PROGRAM RTClock
VAR
	fbGetLocalTime  	: NT_GetTime;
	bBusy				: BOOL;
	bError          	: BOOL :=FALSE;
	nErrID          	: UDINT;
	presetTime      	: TIMESTRUCT;
	syncTimer       	: TON;
	syncTrigger     	: F_TRIG;
	bSynchronize		: BOOL;
	fbRTC_EX2       	: RTC_EX2;
	nMicroseconds   	: DWORD;
	sNetId 				:STRING := '172.16.5.8.1.1';
	LokalClock: STRING(255);
END_VAR

// note: this text did not pass the execution check against the stored diagram
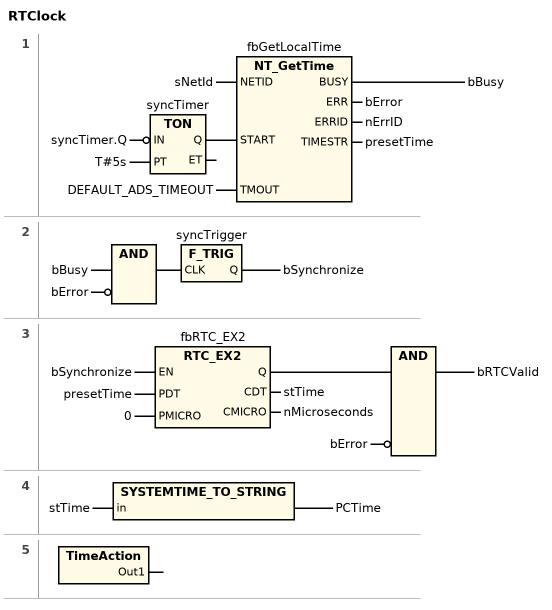
// NETWORK 1
syncTimer(IN := NOT syncTimer.Q, PT := T#5s); // TON
fbGetLocalTime(
    NETID := sNetId,
    START := syncTimer.Q,
    TMOUT := DEFAULT_ADS_TIMEOUT,
    ERR => bError,
    ERRID => nErrID,
    TIMESTR => presetTime); // NT_GetTime
bBusy := fbGetLocalTime.BUSY;

// NETWORK 2
syncTrigger(CLK := bBusy AND NOT bError); // F_TRIG
bSynchronize := syncTrigger.Q;

// NETWORK 3
fbRTC_EX2(EN := bSynchronize, PDT := presetTime, PMICRO := 0, CDT => stTime, CMICRO => nMicroseconds); // RTC_EX2
bRTCValid := fbRTC_EX2.Q AND NOT bError;

// NETWORK 4
PCTime := SYSTEMTIME_TO_STRING(in := stTime);

// NETWORK 5
TimeAction();

ACTION TimeAction:
LokalClock :=DELETE(STR:=PCTime , LEN:=4 , POS:= 20);
IF stTime.wMonth = OldMounth THEN
ChangeOfMounth:= FALSE ;
ELSE
ChangeOfMounth:= TRUE ;
END_IF
IF stTime.wHour = OldHour THEN
bHourChanged := FALSE;
ELSE
bHourChanged:= TRUE;
END_IF
IF stTime.wDay = OldDay THEN
ChangeOfDay := FALSE;
ELSE
ChangeOfDay:= TRUE;
END_IF
IF stTime.wMinute = OldMinute THEN
bMinuteChanged := FALSE ;
ELSE
bMinuteChanged:= TRUE;
END_IF
IF stTime.wHour >17 OR stTime.wHour  <8 THEN
WorkingHour := FALSE;
ELSE
WorkingHour:=TRUE;
END_IF
IF stTime.wDayOfWeek > 0 THEN
ChangeOfweek := TRUE;
ELSE
ChangeOfweek:= FALSE;
END_IF
IF stTime.wDayOfWeek = 0 OR  stTime.wDayOfWeek =  6 THEN
bWeekend := TRUE;
ELSE
bWeekend:= FALSE;
END_IF
END_ACTION

END_PROGRAM

(* stored: Version 1.1.0.1, ProductVersion 3.1.4024.12
   POU RTClock: Id {f41d4fa9-ebc0-48f6-855d-b4f18659f963}, SpecialFunc None
   Action TimeAction: Id {9de085e3-da41-4027-b621-8b242b87b453} *)
